PROGRAM PLC_PRG
VAR
	fbWriteStr						:BFB_WriteStrToFile;
	fbWriteWstr						:BFB_WriteWstrToFile;
END_VAR

fbWriteStr.bBusy

fbWriteWstr.bDone

END_PROGRAM

(* stored: Version 1.1.0.1, ProductVersion 3.1.4024.9
   POU PLC_PRG: Id {f9234ef3-7125-42f2-9743-bf9e8fd2c250}, SpecialFunc None *)
